(* PLC project Sin nombre, Desconocido Sin nombre 1 *)
(* stored: creationDateTime 2024-10-29T16:13:53, modificationDateTime 2024-11-01T19:51:36 *)

PROGRAM program0
  VAR
    CTU0 : CTU;
  END_VAR
  VAR
    BOCINA AT %QX0.0 : BOOL;
    Led1 AT %QX0.1 : BOOL;
    Led2 AT %QX0.2 : BOOL;
    Led3 AT %QX0.3 : BOOL;
    SENSOR_HALL AT %IX0.0 : WORD := 35000;
    pulsador AT %IX0.1 : BOOL;
  END_VAR
  VAR
    RS0 : RS;
    RS1 : DINT;
    TP0 : TP;
    tope_Superior : UINT := 34952;
    tope_Inferior : UINT := 31774;
    in_analogica : WORD := 31800;
    CTU1 : CTU;
    TP1 : TP;
    RS2 : RS;
    SR0 : SR;
    TP2 : TP;
    SR1 : SR;
    SR2 : SR;
    TON0 : TON;
    R_TRIG0 : R_TRIG;
    R_TRIG1 : R_TRIG;
  END_VAR
  VAR  (* added by the conversion: wires and edge detectors of the diagram *)
    _LT19_OUT : BOOL;
    _OR20_OUT : BOOL;
    R_TRIG1_2 : R_TRIG;
    R_TRIG2 : R_TRIG;
    _AND27_OUT : BOOL;
    _AND39_OUT : BOOL;
  END_VAR

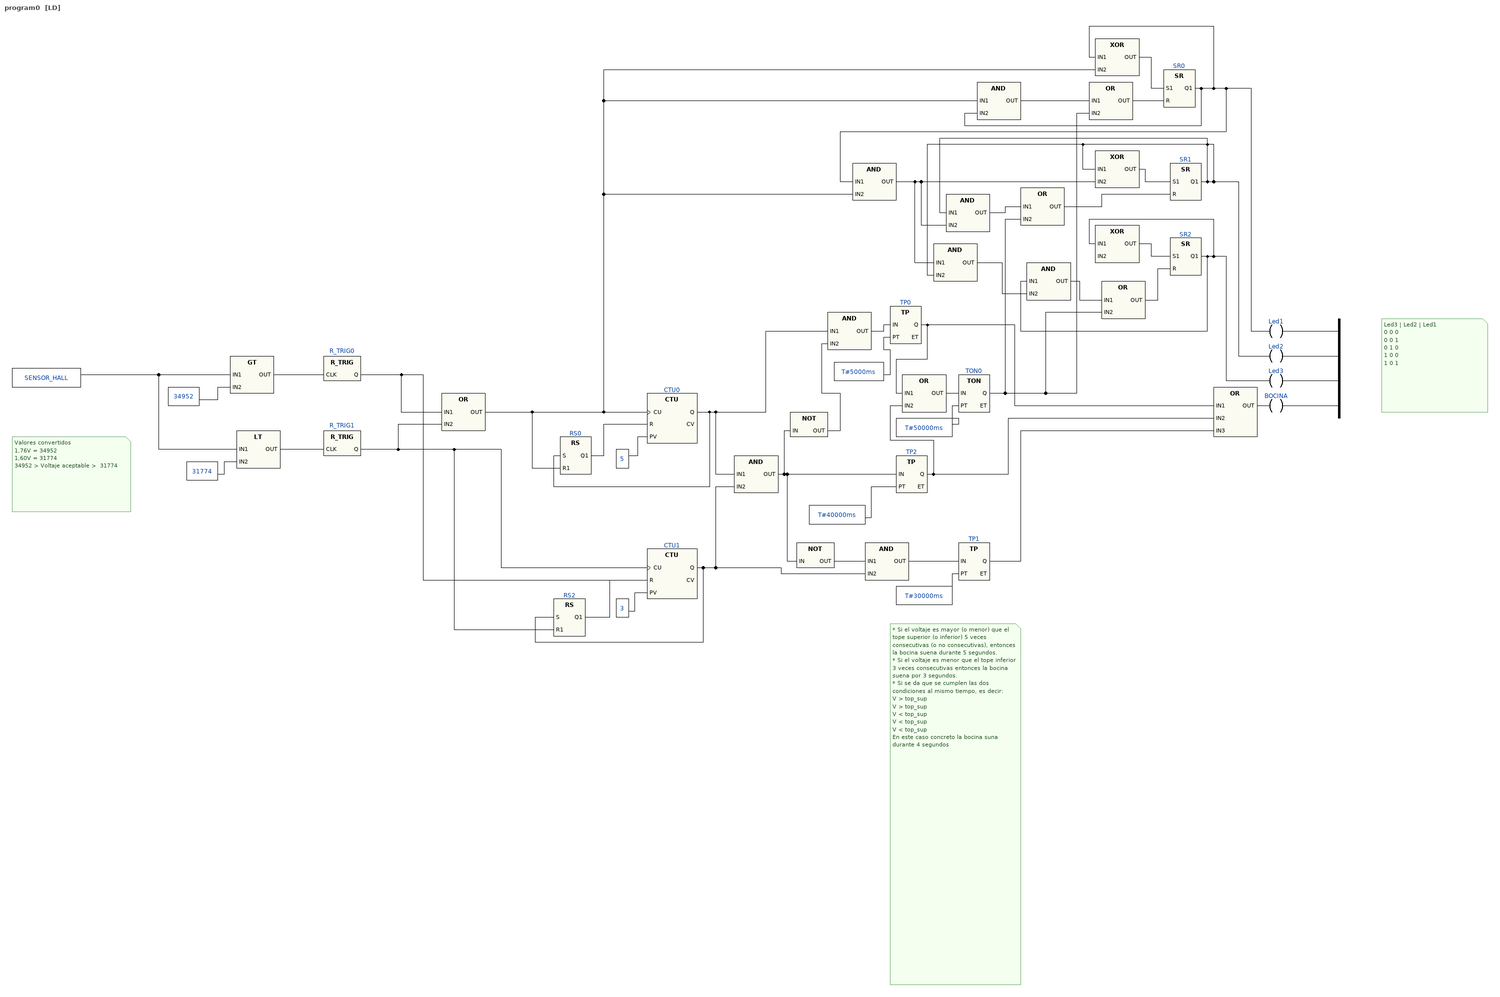
(* LD diagram, written out as Structured Text *)
(* Led3 | Led2 | Led1
0 0 0
0 0 1
0 1 0
1 0 0
1 0 1 *)
R_TRIG0(CLK := SENSOR_HALL > 34952);
_LT19_OUT := SENSOR_HALL < 31774;
R_TRIG1(CLK := _LT19_OUT);
_OR20_OUT := R_TRIG0.Q OR R_TRIG1.Q;
R_TRIG1_2(CLK := _OR20_OUT);
RS0(S := CTU0.Q, R1 := _OR20_OUT);
CTU0(CU := R_TRIG1_2.Q, R := RS0.Q1, PV := 5);
R_TRIG2(CLK := R_TRIG1.Q);
RS2(S := CTU1.Q, R1 := R_TRIG1.Q);
CTU1(CU := R_TRIG2.Q, R := RS2.Q1 OR R_TRIG0.Q, PV := 3);
_AND27_OUT := CTU0.Q AND CTU1.Q;
TP0(IN := CTU0.Q AND NOT _AND27_OUT, PT := T#5000ms);
TP2(IN := _AND27_OUT, PT := T#40000ms);
TP1(IN := NOT _AND27_OUT AND CTU1.Q, PT := T#30000ms);
BOCINA := TP0.Q OR TP2.Q OR TP1.Q;
TON0(IN := TP0.Q OR TP2.Q, PT := T#50000ms);
SR0(S1 := SR0.Q1 XOR _OR20_OUT, R := _OR20_OUT AND SR0.Q1 OR TON0.Q);
Led1 := SR0.Q1;
_AND39_OUT := SR0.Q1 AND _OR20_OUT;
SR1(S1 := SR1.Q1 XOR _AND39_OUT, R := SR1.Q1 AND _AND39_OUT OR TON0.Q);
Led2 := SR1.Q1;
SR2(S1 := XOR(IN1 := SR2.Q1), R := SR2.Q1 AND _AND39_OUT AND SR1.Q1 OR TON0.Q);
Led3 := SR2.Q1;
(* Valores convertidos 
1,76V = 34952
1,60V = 31774
34952 > Voltaje aceptable >  31774 *)
(* * Si el voltaje es mayor (o menor) que el tope superior (o inferior) 5 veces consecutivas (o no consecutivas), entonces la bocina suena durante 5 segundos.
* Si el voltaje es menor que el tope inferior 3 veces consecutivas entonces la bocina suena por 3 segundos.
* Si se da que se cumplen las dos condiciones al mismo tiempo, es decir:
V > top_sup
V > top_sup
V < top_sup
V < top_sup
V < top_sup
En este caso concreto la bocina suna durante 4 segundos *)
END_PROGRAM

CONFIGURATION Config0
  RESOURCE Res0 ON PLC
    TASK task0(INTERVAL := T#20ms, PRIORITY := 0);
    PROGRAM instance0 WITH task0 : program0;
  END_RESOURCE
END_CONFIGURATION
